// TwinCAT 3 PLC project Untitled1
// ProgramVersion: 3.1.4026.16
// CompilerDefines: VISU_USEPROPERTYINFO
// libraries:
//   Tc2_Standard, * (Beckhoff Automation GmbH)
//   Tc2_System, * (Beckhoff Automation GmbH)
//   VisuSymbols, 4.5.0.0 (System)
// project tree:
//   / GlobalTextList.TcGTLO, PlcTask.TcTTO, Visualization Manager.TcVMO (not stored)
//   POUs/ MAIN.TcPOU
//   VISUs/ Visualization.TcVIS
// real-time tasks:
//   TASK PlcTask: cycle T#10ms, priority 20, ADS port 350

CONFIGURATION Untitled1
    RESOURCE PLC ON TwinCAT3
        TASK PlcTask(INTERVAL := T#10ms, PRIORITY := 20);
        PROGRAM MAIN WITH PlcTask : MAIN;
    END_RESOURCE
END_CONFIGURATION

// ---- POUs/MAIN.TcPOU
PROGRAM MAIN
VAR
	rAngle : REAL;
	rAngularVelocity : REAL := 60;
	rRadius : REAL := 80;
	rStickLength : REAL := 100;
	rDistance : REAL;
	rLength : REAL;
	pi : REAL := 3.14159265;
	
	ip1x : REAL;
	ip1y : REAL;
	ip2x : REAL;
	ip2y : REAL;
END_VAR

IF rRadius > rStickLength THEN
	rRadius := rStickLength;
END_IF

rAngle := rAngle + rAngularVelocity * 0.01;

rLength := (1-COS(rAngle * (pi / 180))) * rRadius + SQRT((rStickLength * rStickLength) - (rRadius * rRadius * SIN(rAngle * (pi / 180)) * SIN(rAngle * (pi / 180))));
rDistance := rLength - rStickLength;

ip1x := COS(rAngle * (pi / 180)) * rRadius * -1;
ip1y := SIN(rAngle * (pi / 180)) * rRadius;

ip2x := rLength - rRadius;
ip2y := 0;

END_PROGRAM

// ---- VISUs/Visualization.TcVIS
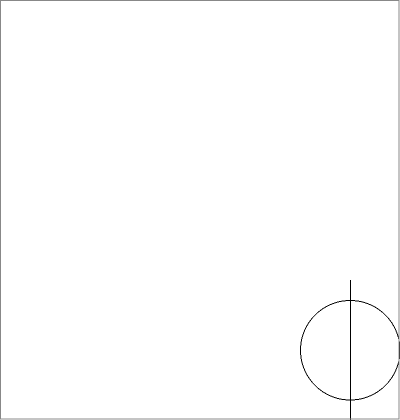
VISUALIZATION Visualization  // 400x420
    Ellipse (300,300 100x100)
        p1097714728: MAIN.rRadius * 20
    Line (350,350) (350,350)
        p3528305787: MAIN.ip1x
        p2773130477: MAIN.ip1y
        p874137650: MAIN.ip2x
        p1126004900: MAIN.ip2y
    Line (350,300) (350,420)
        p3528305787: MAIN.rStickLength + MAIN.rRadius
        p874137650: MAIN.rStickLength + MAIN.rRadius
    Line (350,280) (350,400)
        p3528305787: MAIN.rStickLength - MAIN.rRadius
        p874137650: MAIN.rStickLength - MAIN.rRadius
END_VISUALIZATION
